Staubli VAL3: OnF1.pgx

program OnF1()
begin
  //原始文件
  call RobMaster:start()
  bUserRefresh=true
end
